TYPE ST_Part :
STRUCT
	runningNumber	: INT;
	variant			: INT;
	ID				: STRING;
	timeStamp		: INT;
	route			: INT;
	scrap			: BOOL;
	jobs			: DINT;
	user			: STU_Part;
END_STRUCT
END_TYPE

(* stored: Version 1.1.0.1
   DUT ST_Part: Id {44a23a29-eb4c-4438-b72b-70c47db83b22} *)
